{attribute 'qualified_only'}
{attribute 'strict'}
TYPE SensorBrands :
(
	Sick,
	Pliz,
	Parker,
	Bosch
);
END_TYPE

(* stored: Version 1.1.0.1, ProductVersion 3.1.4024.12
   DUT SensorBrands: Id {bd54fced-0772-4f7a-914b-23bbb176ed37} *)
